
// ===== library: MasterCopy "Start_Stop" =====

VAR_GLOBAL   // PLC tag table "Start_Stop"
   "IX_START" AT %I4.4 : Bool;
   "IX_STOP" AT %I4.6 : Bool;
END_VAR

// ===== library: MasterCopy "SSC - Sensor-Station" =====

VAR_GLOBAL   // PLC tag table "SSC - Sensor-Station"
   "QX_SSC_LED_Green_Q5" AT %Q6.4 : Bool;
   "QX_SSC_LED_Yellow_Q6" AT %Q6.5 : Bool;
   "QX_SSC_LED_Red_Q7" AT %Q6.6 : Bool;
   "QX_SSC_LED_Red_Online_Q8" AT %Q6.7 : Bool;
   "IX_SSC_LightBarrierStorage_I3" AT %I4.3 : Bool;
   "IX_SSC_LightBarrierOutsourcing_I4" AT %I4.2 : Bool;
   "IW_SSC_ColorSensor_A1" AT %IW9 : Word;
END_VAR

// ===== library: MasterCopy "SLD - Sorting Line with Detection" =====

VAR_GLOBAL   // PLC tag table "SLD - Sorting Line with Detection"
   "IX_SLD_PulseCounter_I1" AT %I3.0 : Bool;
   "IX_SLD_LightBarrierInlet_I2" AT %I3.1 : Bool;
   "IX_SLD_LightBarrierBehindColorSensor_I3" AT %I3.2 : Bool;
   "IW_SLD_ColorSensor_A4" AT %IW7 : Word;
   "IX_SLD_LightBarrierWhite_I5" AT %I3.3 : Bool;
   "IX_SLD_LightBarrierRed_I6" AT %I3.4 : Bool;
   "IX_SLD_LightBarrierBlue_I7" AT %I3.5 : Bool;
   "QX_SLD_M1_ConveyorBelt_Q1" AT %Q5.0 : Bool;
   "QX_SLD_Compressor_Q2" AT %Q5.1 : Bool;
   "QX_SLD_ValveFirstEjectorWhite_Q3" AT %Q5.2 : Bool;
   "QX_SLD_ValveSecondEjectorRed_Q4" AT %Q5.3 : Bool;
   "QX_SLD_ValveThirdEjectorBlue_Q5" AT %Q5.4 : Bool;
END_VAR

// ===== library: MasterCopy "VGR - Vacuum Gripper Robot" =====

VAR_GLOBAL   // PLC tag table "VGR - Vacuum Gripper Robot"
   "IX_VGR_RefSwitchVerticalAxis_I1" AT %I1.6 : Bool;
   "IX_VGR_RefSwitchHorizontalAxis_I2" AT %I3.6 : Bool;
   "IX_VGR_RefSwitchRotate_I3" AT %I3.7 : Bool;
   "IX_VGR_EncoderVerticalAxisImp1_B1" AT %I6.0 : Bool;
   "IX_VGR_EncoderVerticalAxisImp2_B2" AT %I6.4 : Bool;
   "IX_VGR_EncoderHorizontalAxisImp1_B3" AT %I6.1 : Bool;
   "IX_VGR_EncoderHorizontalAxisImp2_B4" AT %I6.5 : Bool;
   "IX_VGR_EncoderRotateImp1_B5" AT %I6.2 : Bool;
   "IX_VGR_EncoderRotateImp2_B6" AT %I6.6 : Bool;
   "QX_VGR_M1_VerticalAxisUp_Q1" AT %Q2.0 : Bool;
   "QX_VGR_M1_VerticalAxisDown_Q2" AT %Q2.1 : Bool;
   "QX_VGR_M2_HorizontalAxisBackward_Q3" AT %Q2.2 : Bool;
   "QX_VGR_M2_HorizontalAxisForward_Q4" AT %Q2.3 : Bool;
   "QX_VGR_M3_RotateClockwise_Q5" AT %Q2.4 : Bool;
   "QX_VGR_M3_RotateCounterclockwise_Q6" AT %Q2.5 : Bool;
   "QX_VGR_Compressor_Q7" AT %Q2.6 : Bool;
   "QX_VGR_ValveVacuum_Q8" AT %Q2.7 : Bool;
   "QW_VGR_PWM_Vertical_M1" AT %QW15 : Int;
   "QW_VGR_PWM_Horizontal_M2" AT %QW17 : Int;
   "QW_VGR_PWM_Rotate_M3" AT %QW19 : Int;
END_VAR

// ===== library: MasterCopy "SSC - Camera-Station" =====

VAR_GLOBAL   // PLC tag table "SSC - Camera-Station"
   "IX_SSC_RefSwitchVerticalAxis_I1" AT %I4.0 : Bool;
   "IX_SSC_RefSwitchHorizontalAxis_I2" AT %I4.1 : Bool;
   "IX_SSC_EncoderVerticalAxisImp1_B1" AT %I5.3 : Bool;
   "IX_SSC_EncoderVerticalAxisImp2_B2" AT %I5.7 : Bool;
   "IX_SSC_EncoderHorizontalAxisImp1_B3" AT %I6.3 : Bool;
   "IX_SSC_EncoderHorizontalAxisImp2_B4" AT %I6.7 : Bool;
   "QX_SSC_M1_VerticalAxisUp_Q1" AT %Q6.0 : Bool;
   "QX_SSC_M1_VerticalAxisDown_Q2" AT %Q6.1 : Bool;
   "QX_SSC_M2_HorizontalAxisClockwise_Q3" AT %Q6.3 : Bool;
   "QX_SSC_M2_HorizontalAxisCounterclockwise_Q4" AT %Q6.2 : Bool;
   "QW_SSC_PWM_Vertical_M1" AT %QW27 : Int;
   "QW_SSC_PWM_Horizontal_M2" AT %QW29 : Int;
END_VAR

// ===== library: MasterCopy "MPO - Multi Processing Station with Oven" =====

VAR_GLOBAL   // PLC tag table "MPO - Multi Processing Station with Oven"
   "IX_MPO_RefSwitchTurnTable_PosVac_I1" AT %I1.7 : Bool;
   "IX_MPO_RefSwitchTurnTable_PosBelt_I2" AT %I2.0 : Bool;
   "IX_MPO_LightBarrierEndOfConBelt_I3" AT %I2.1 : Bool;
   "IX_MPO_RefSwitchTurnTable_PosSaw_I4" AT %I2.2 : Bool;
   "IX_MPO_RefSwitchVac_PosTurnTable_I5" AT %I2.3 : Bool;
   "IX_MPO_RefSwitchOvenFeederInside_I6" AT %I2.4 : Bool;
   "IX_MPO_RefSwitchOvenFeederOutside_I7" AT %I2.5 : Bool;
   "IX_MPO_RefSwitchVac_PosOven_I8" AT %I2.6 : Bool;
   "IX_MPO_LightBarrierOven_I9" AT %I2.7 : Bool;
   "QX_MPO_M1_TurnTableClockwise_Q1" AT %Q3.0 : Bool;
   "QX_MPO_M1_TurnTableCounterclockwise_Q2" AT %Q3.1 : Bool;
   "QX_MPO_M2_ConveyorBeltForward_Q3" AT %Q3.2 : Bool;
   "QX_MPO_M3_Saw_Q4" AT %Q3.3 : Bool;
   "QX_MPO_M4_OvenFeederRetract_Q5" AT %Q3.4 : Bool;
   "QX_MPO_M4_OvenFeederExtend_Q6" AT %Q3.5 : Bool;
   "QX_MPO_M5_VacuumTowardsOven_Q7" AT %Q3.6 : Bool;
   "QX_MPO_M5_VacuumTowardsTurnTable_Q8" AT %Q3.7 : Bool;
   "QX_MPO_LightOven_Q9" AT %Q4.0 : Bool;
   "QX_MPO_Compressor_Q10" AT %Q4.1 : Bool;
   "QX_MPO_ValveVacuum_Q11" AT %Q4.2 : Bool;
   "QX_MPO_ValveLowering_Q12" AT %Q4.3 : Bool;
   "QX_MPO_ValveOvenDoor_Q13" AT %Q4.4 : Bool;
   "QX_MPO_ValveFeeder_Q14" AT %Q4.5 : Bool;
   "QW_MPO_PWM_TurnTable_M1" AT %QW23 : Int;
   "QW_MPO_PWM_Vacuum_M5" AT %QW25 : Int;
END_VAR

// ===== library: MasterCopy "HBW - Automated High-Bay Warehouse" =====

VAR_GLOBAL   // PLC tag table "HBW - Automated High-Bay Warehouse"
   "IX_HBW_RefSwitchHorizontalAxis_I1" AT %I1.0 : Bool;
   "IX_HBW_LightBarrierInside_I2" AT %I1.1 : Bool;
   "IX_HBW_LightBarrierOutside_I3" AT %I1.2 : Bool;
   "IX_HBW_RefSwitchVerticalAxis_I4" AT %I1.3 : Bool;
   "IX_HBW_TrailSensor1Lower_A1" AT %I5.0 : Bool;
   "IX_HBW_TrailSensor2Upper_A2" AT %I5.4 : Bool;
   "IX_HBW_EncoderVerticalAxisImp1_B3" AT %I5.2 : Bool;
   "IX_HBW_EncoderVerticalAxisImp2_B4" AT %I5.6 : Bool;
   "IX_HBW_EncoderHorizontalAxisImp1_B1" AT %I5.1 : Bool;
   "IX_HBW_EncoderHorizontalAxisImp2_B2" AT %I5.5 : Bool;
   "IX_HBW_SwitchCantileverFront_I5" AT %I1.4 : Bool;
   "IX_HBW_SwitchCantileverBack_I6" AT %I1.5 : Bool;
   "QX_HBW_M1_ConveyorBeltForward_Q1" AT %Q1.0 : Bool;
   "QX_HBW_M1_ConveyorBeltBackward_Q2" AT %Q1.1 : Bool;
   "QX_HBW_M2_HorizontalTowardsRack_Q3" AT %Q1.2 : Bool;
   "QX_HBW_M2_HorizontalTowardsConveyorBelt_Q4" AT %Q1.3 : Bool;
   "QX_HBW_M3_VerticalAxisDownward_Q5" AT %Q1.4 : Bool;
   "QX_HBW_M3_VerticalAxisUpward_Q6" AT %Q1.5 : Bool;
   "QX_HBW_M4_CantileverForward_Q7" AT %Q1.6 : Bool;
   "QX_HBW_M4_CantileverBackward_Q8" AT %Q1.7 : Bool;
   "QW_HBW_PWM_ConveyorBelt_M1" AT %QW7 : Int;
   "QW_HBW_PWM_HorizontalAxis_M2" AT %QW9 : Int;
   "QW_HBW_PWM_VerticalAxis_M3" AT %QW11 : Int;
   "QW_HBW_PWM_Cantilever_M4" AT %QW13 : Int;
END_VAR

// ===== library: MasterCopy "FB_INC_DEC" =====

// folder: Positioning

FUNCTION_BLOCK "FB_INC_DEC"   // FB9, SCL
TITLE = position with encoder
{ S7_Optimized_Access := 'TRUE' }
VERSION : 0.1
   VAR_INPUT
      inx_CHa : Bool := false;   // Encoder impulse 2 channel a / Encoderimpulse 2 Kanal a
      inx_CHb : Bool := false;   // Encoder impulse 1 channel b / / Encoderimpulse 1 Kanal b
      inx_RST : Bool := False;   // Reference switch / Referenzpunkt
      ini_Ref_val : Int := 0;   // Reference value / Referenzwert
   END_VAR
   VAR_OUTPUT
      outx_dir : Bool := false;   // direction / Richtung
      outi_cnt : Int := 0;   // position / Position
   END_VAR
   VAR
      lx_edgea : Bool := False;
      lx_clka : Bool;
      lx_clkb : Bool;
      lx_edgeb : Bool;
      lx_axb : Bool;
      lx_dir : Bool;
      li_cnt : Int;
   END_VAR
BEGIN

   #lx_axb := #inx_CHa XOR #inx_CHb;

   (* create pulses for channel a *)
   #lx_clka := #inx_CHa XOR #lx_edgea;
   #lx_edgea := #inx_CHa;

   (* create pulses for channel b *)
   #lx_clkb := #inx_CHb XOR #lx_edgeb;
   #lx_edgeb := #inx_CHb;

   (* create pulses for both channels *)
   #lx_clka := #lx_clka OR #lx_clkb;

   (* set the direction output *)
   IF #lx_axb AND #lx_clka THEN
       #lx_dir := TRUE;
   END_IF;
   IF #lx_axb AND #lx_clkb THEN
       #lx_dir := FALSE;
   END_IF;

   (* increment or decrement the counter *)
   IF #lx_clka AND #lx_dir THEN
       #li_cnt := #li_cnt + 1;
   END_IF;
   IF #lx_clka AND NOT #lx_dir THEN
       #li_cnt := #li_cnt - 1;
   END_IF;

   (* reset the counter if rst active *)
   IF #inx_RST THEN
       #li_cnt := #ini_Ref_val;
   END_IF;

   #outx_dir := #lx_dir;
   #outi_cnt := #li_cnt;
END_FUNCTION_BLOCK